PROGRAM MAIN
VAR
	fbEventLoggerListener : FB_EventLoggerListenerImpl;
	aLoggedEvents : ARRAY[0..99] OF ST_LoggedEvent;
END_VAR



fbEventLoggerListener(aLoggedEventsBuffer:= aLoggedEvents);

END_PROGRAM

(* stored: Version 1.1.0.1, ProductVersion 3.1.4024.12
   POU MAIN: Id {b456ed00-d5bf-423c-93f9-9669130ca655}, SpecialFunc None *)
